// Mitsubishi GX Works2 project: silEx2   PLC: Q03UDV

PROGRAM MAIN
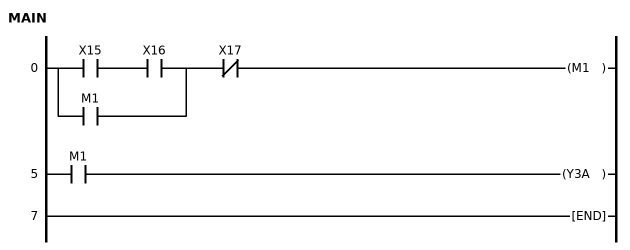
0     LD      X15
      AND     X16
      OR      M1
      ANI     X17
      OUT     M1
5     LD      M1
      OUT     Y3A
7     END
END_PROGRAM
